(* CoDeSys 2.3 export: ST_ISSUESPECIFICTYPES.EXP *)

(* Data type *)
TYPE ST_IssueSpecificTypes :
STRUCT
	Issue94	: ST_Issue94;
END_STRUCT
END_TYPE
